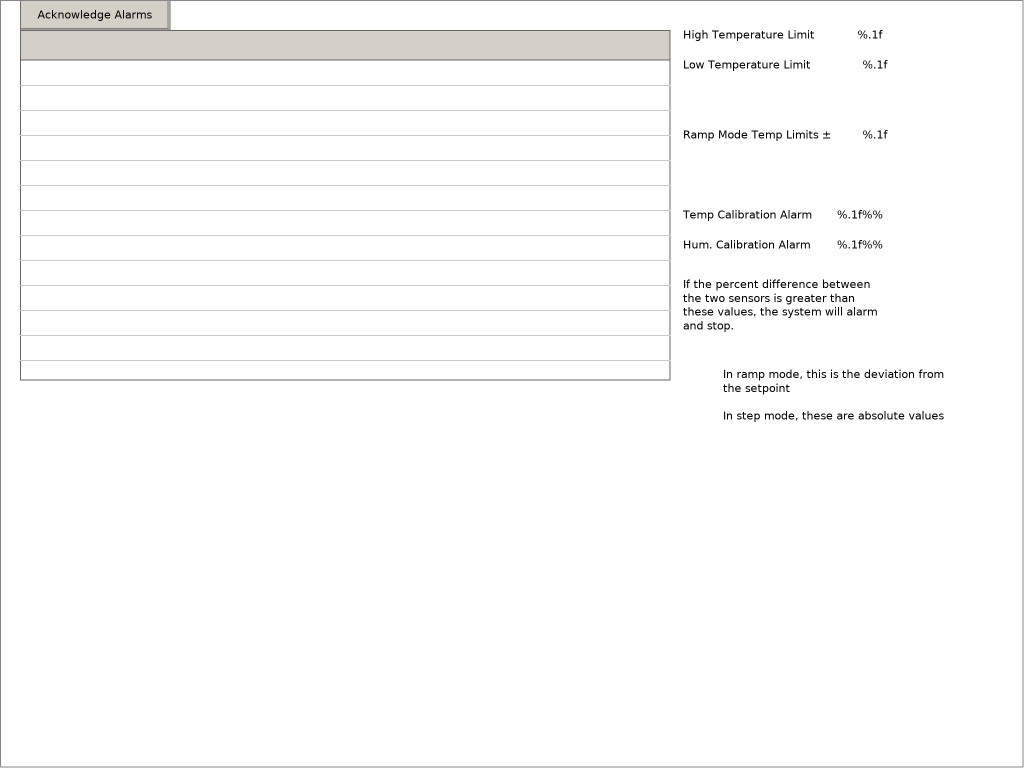
VISUALIZATION Alarms  // 1024x768
    Table (20,30 650x350), data array: GVL.aAlarms
        p511219082: Alarm Note
        p1892666644: GVL.aAlarms[INDEX].sAlarmText
        p2232123230: Date & Time
        p3854506369: GVL.aAlarms[INDEX].dtTime
    Textfield (840,20 60x30), "%.1f", text variable: GVL.TempAlarmHigh
        OnMouseClick: write the text variable via VisuDialogs.Numpad, min -10, max 50
    Label (680,20 150x30), "High Temperature Limit"
    Textfield (840,50 70x30), "%.1f", text variable: GVL.TempAlarmLow
        OnMouseClick: write the text variable via VisuDialogs.Numpad, min -10, max 50
    Label (680,50 150x30), "Low Temperature Limit"
    Button (20,0 150x30), "Acknowledge Alarms", colour toggle: GVL.bActiveAlarm
        OnMouseClick: execute { GVL.bActiveAlarm:=FALSE; }
    Textfield (720,360 260x70), "In ramp mode, this is the deviation from the setpoint In step mode, these are absolute values"
    Textfield (810,200 100x30), "%.1f%%", text variable: GVL.TempCalibrationLimit
        OnMouseClick: write the text variable via Default, min 1, max 100
    Label (680,200 150x30), "Temp Calibration Alarm"
    Textfield (810,230 100x30), "%.1f%%", text variable: GVL.HumCalibrationLimit
        OnMouseClick: write the text variable via VisuDialogs.Numpad, min 1, max 100
    Label (680,230 150x30), "Hum. Calibration Alarm"
    Textfield (680,270 260x70), "If the percent difference between the two sensors is greater than these values, the system will alarm and stop."
    Label (680,120 150x30), "Ramp Mode Temp Limits ±"
    Textfield (840,120 70x30), "%.1f", text variable: GVL.TempRampModeAlarm
        OnMouseClick: write the text variable via VisuDialogs.Numpad, min -10, max 50
END_VISUALIZATION

(* stored: Version 1.1.0.1, ProductVersion 3.1.4022.18
   Visu Alarms: Id {15a5794a-8e40-49e4-852c-b1a0ebfe9cc1} *)
